FUNCTION FC_WriteProgLine : BOOL
VAR_INPUT
	sLine			: STRING(MAX_STRING_LENGTH);	// GeoCode Befehl
END_VAR
VAR
END_VAR

IF GVL_HexaBridge.bHexConnected AND GVL_HexaBridge.bBridgeRunning THEN
	// Senden des Befehls
	IF GVL_HexaBridge.sProgLine = '' AND NOT GVL_HexaBridge.bProgLineReady AND GVL_HexaBridge.bProgLineSaved
	AND NOT GVL_HexaBridge.bExecute AND NOT GVL_HexaBridge.bProgLineExecution THEN
		GVL_HexaBridge.bProgLineSaved := FALSE;
		GVL_HexaBridge.sProgLine := sLine;
		GVL_HexaBridge.bProgLineReady := TRUE;
		FC_WriteProgLine := TRUE;
	END_IF
END_IF

END_FUNCTION

(* stored: Version 1.1.0.1
   POU FC_WriteProgLine: Id {adf96a24-e6c6-463b-91f4-0a8a4fb38158}, SpecialFunc None *)
